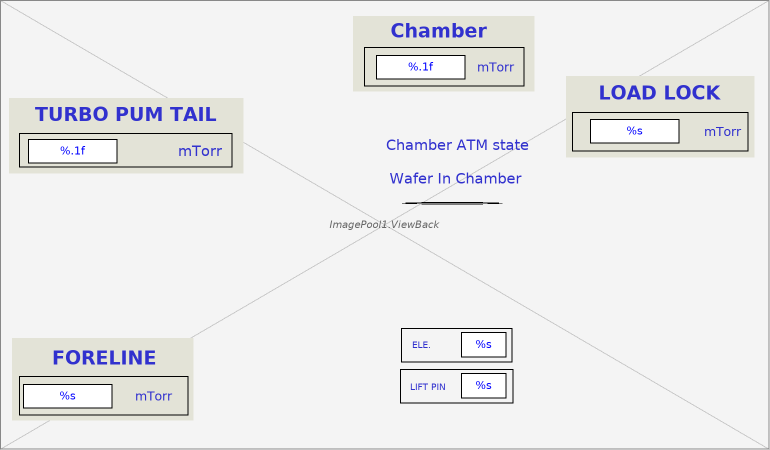
VISUALIZATION ViewPar_1  // 770x450
    Image (0,0 769x449), image: ImagePool1.ViewBack
    Label (361,129 193x32), "Chamber ATM state", invisible if: NOT gICP.I_ATMSensor
    Group (566,76 188x81)
        RoundedRectangle (0,0 188x81)
        Label (12,1 163x32), "LOAD LOCK"
        RoundedRectangle (6,36 176x39)
        RoundedRectangle (24,43 89x24), "%s", text variable: gICP.LoadLockGauge.outputValue_String, colour toggle: gICP.LoadLockGauge.error
        Label (135,44 41x23), "mTorr"
    Group (353,16 181x75)
        RoundedRectangle (0,0 181x75)
        Label (14,2 150x26), "Chamber"
        Label (121,40 50x22), "mTorr"
        RoundedRectangle (23,39 89x24), "%.1f", text variable: gICP.ChamberGauge.outputValue1, colour toggle: gICP.ForeLineGauge.error
        RoundedRectangle (11,31 160x39)
    RoundedRectangle (12,338 181x82)
    Label (39,341 131x34), "FORELINE"
    Label (132,385 50x22), "mTorr"
    RoundedRectangle (23,384 89x24), "%s", text variable: gICP.ForeLineGauge.outputValue_String, colour toggle: gICP.ForeLineGauge.error
    RoundedRectangle (19,376 169x39)
    Group (9,98 234x75)
        RoundedRectangle (0,0 234x75)
        Label (11,2 212x29), "TURBO PUM TAIL"
        Label (166,42 50x22), "mTorr"
        RoundedRectangle (19,41 89x24), "%.1f", text variable: gICP.TBGauge.outputValue, colour toggle: gICP.TBGauge.error
        RoundedRectangle (10,35 213x34)
    Ellipse (402,202 100x2), colour toggle: gWaferMemoryState=1
        OnMouseClick: execute { gWaferMemoryState:=BOOL_TO_INT(NOT INT_TO_BOOL(gWaferMemoryState)); ups_CX51X0.Act_Wrtie(); }
    Label (384,166 143x25), "Wafer In Chamber", invisible if: NOT otherMachineState.lightShow
    RoundedRectangle (401,328 111x34)
    Label (409,335 28x20), "ELE."
    RoundedRectangle (400,369 113x34)
    Label (407,377 50x20), "LIFT PIN"
    RoundedRectangle (461,332 45x25), "%s", text variable: gICP.ElectrodeCyl.HMIItf.sensorShow
    RoundedRectangle (461,373 45x25), "%s", text variable: gICP.LiftPinCyl.HMIItf.sensorShow
END_VISUALIZATION

(* stored: Version 1.1.0.1, ProductVersion 3.1.4024.12
   Visu ViewPar_1: Id {ca517d0e-512e-46dd-a24a-23b145b93d1f} *)
